INTERFACE ITF_Regelschuif_OutClose_DG

METHOD set : BOOL
VAR_INPUT
	state : BOOL;	
END_VAR
END_METHOD

END_INTERFACE

(* stored: Version 1.1.0.1, ProductVersion 3.1.4026.8
   Itf ITF_Regelschuif_OutClose_DG: Id {d4dd24ca-4a3f-4e66-aaf3-3c7a7c648480}
   Method set: Id {95353664-ab06-49ba-a9ce-f275afa138e2} *)
